// TIA Portal V19 export
VAR_GLOBAL   // PLC tag table "CentralFunctions"
END_VAR
